// TIA Portal V20 export
FUNCTION "Startup_FC" : Void   // FC1, LAD
{ S7_Optimized_Access := 'TRUE' }
// stored: SetENOAutomatically false
   VAR_TEMP
      ResetCount_0 : DInt;
      ResetCount_1 : DInt;
      P_Trig : Bool;
   END_VAR
   VAR_TEMP   // added for the SCL form of the ladder/FBD networks
      _w1 : Bool;
   END_VAR
BEGIN

REGION Network 1
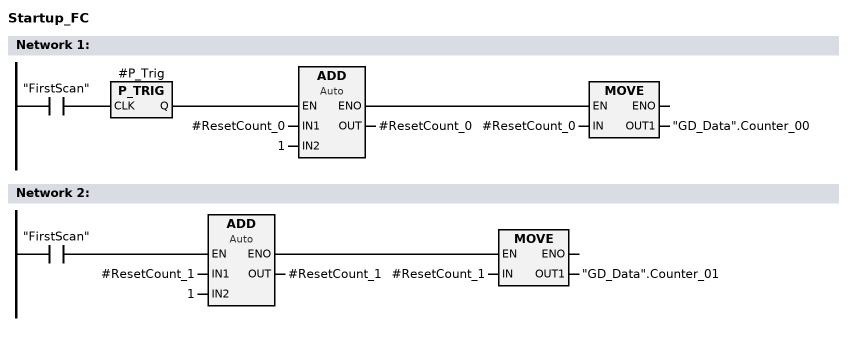
   RUNG wire#powerrail
      Contact( "FirstScan" )
      P_Trig( #P_Trig )
      { S7_GenerateENO := "TRUE" } Add(in1 := #ResetCount_0, in2 := 1, out => #ResetCount_0)
      { S7_GenerateENO := "TRUE" } Move(in := #ResetCount_0, out1 => "GD_Data".Counter_00)
   END_RUNG
   // the same network as SCL:
   // ENO of a box is taken as its EN; it also drops when the box reports an error
   #_w1 := "FirstScan" AND NOT #P_Trig;   // rising edge
   #P_Trig := "FirstScan";
   IF #_w1 THEN
       #ResetCount_0 := #ResetCount_0 + 1;
       "GD_Data".Counter_00 := #ResetCount_0;
   END_IF;
END_REGION

REGION Network 2
   RUNG wire#powerrail
      Contact( "FirstScan" )
      { S7_GenerateENO := "TRUE" } Add(in1 := #ResetCount_1, in2 := 1, out => #ResetCount_1)
      { S7_GenerateENO := "TRUE" } Move(in := #ResetCount_1, out1 => "GD_Data".Counter_01)
   END_RUNG
   // the same network as SCL:
   // ENO of a box is taken as its EN; it also drops when the box reports an error
   IF "FirstScan" THEN
       #ResetCount_1 := #ResetCount_1 + 1;
       "GD_Data".Counter_01 := #ResetCount_1;
   END_IF;
END_REGION
END_FUNCTION
